{attribute addProperty BoxType "EJ7211-0011-0026"}
{attribute addProperty Id "Target_velocityAT %Q*DINT324"}
{attribute addProperty CRC "1403554480"}
{attribute addProperty SizeInBites "32"}
{attribute addProperty SizeInBytes "4"}
TYPE DS402_Target_velocity_53A88AB0 :
STRUCT
	{attribute addProperty Name "Target_velocity"}
	Target_velocity AT %Q* : DINT;
END_STRUCT
END_TYPE

(* stored: Version 1.2.0.0, ProductVersion 3.1.4024.9
   DUT DS402_Target_velocity_53A88AB0: Id {ad05e6de-14e5-4bee-acb9-3a311681535a} *)
